Yaskawa INFORM job: test_long.JBI

version: 0
/JOB
//NAME test_long
//POS
///NPOS 48,0,0,2,0,0
///TOOL 1
///POSTYPE ROBOT
///RECTAN
///RCONF 1,0,0,0,0,0,0,0,0,0,0,0,0,0,0,0,0,0,0,0,0,0,0,0
//INST
///DATE 03/29/2021 17:02
///COMM
///ATTR SC,RW
///FRAME ROBOT
///GROUP1 RB1
NOP
CALL JOB:DEBUT
'Part trajectory number: 0
CALL JOB:test_long_tjr0
'Part trajectory number: 1
CALL JOB:test_long_tjr1
'Part trajectory number: 2
CALL JOB:test_long_tjr2
'Part trajectory number: 3
CALL JOB:test_long_tjr3
'Part trajectory number: 4
CALL JOB:test_long_tjr4
'Part trajectory number: 5
CALL JOB:test_long_tjr5
'Part trajectory number: 6
CALL JOB:test_long_tjr6
'Part trajectory number: 7
CALL JOB:test_long_tjr7
CALL JOB:FIN
END
